// TIA Portal V19 export
DATA_BLOCK "Encoder"   // DB160
{ S7_Optimized_Access := 'TRUE' }
// stored: MemoryReserve 100
   VAR
      "1248A1" { S7_SetPoint := 'True'} : PD_TEL81;   // Encoder lineare su pinza misuratore calcolo FAK
   END_VAR
BEGIN
END_DATA_BLOCK
